// TIA Portal project "MPS1.1" (V16)

(* hardware
DEVICE "S7-1200 station_1"  S7-1200 Station
   slot 0: "Rack_0"  S7-1200 Rack  Rack  V1.0
   slot 1: "PLC_1"  CPU 1214C DC/DC/DC  6ES7 214-1AG40-0XB0  V4.4
   slot 2: "DI 8/DQ 8x24VDC_1"  6ES7 223-1BH32-0XB0  V2.0
*)

// ===== PLC "PLC_1"  CPU 1214C DC/DC/DC =====

VAR_GLOBAL   // PLC tag table "Default tag table"
   "System_Byte" AT %MB1 : Byte;
   "FirstScan" AT %M1.0 : Bool;
   "DiagStatusUpdate" AT %M1.1 : Bool;
   "AlwaysTRUE" AT %M1.2 : Bool;
   "AlwaysFALSE" AT %M1.3 : Bool;
   "Start NO" AT %I0.0 : Bool;
   "Stop NC" AT %I0.1 : Bool;
   "Reset NO" AT %I0.2 : Bool;
   "M/A Seletor" AT %I0.3 : Bool;
   "C2BG1" AT %I0.5 : Bool;
   "C2BG2" AT %I0.6 : Bool;
   "PART-AV1" AT %I0.7 : Bool;
   "C2BG3 NC" AT %I1.0 : Bool;
   "G1BG1 NO" AT %I1.1 : Bool;
   "G1BG2 NO" AT %I1.2 : Bool;
   "G1BG3 NC" AT %I1.3 : Bool;
   "Emergência NC" AT %I1.4 : Bool;
   "Pressostato NC" AT %I1.5 : Bool;
   "LED Start" AT %Q0.0 : Bool;
   "LED Reset" AT %Q0.1 : Bool;
   "Luz Q1" AT %Q0.2 : Bool;
   "Luz Q2" AT %Q0.3 : Bool;
   "Conv. anda p/ dir." AT %Q0.4 : Bool;
   "Conv. anda p/ esq." AT %Q0.5 : Bool;
   "Av. Cil. Alim." AT %Q0.6 : Bool;
   "Seletor Conv." AT %Q0.7 : Bool;
   "Válvula NC" AT %Q1.0 : Bool;
   "T1_STATUS" AT %M0.0 : Bool;
   "T2_STATUS" AT %M0.1 : Bool;
   "T3_STATUS" AT %M0.2 : Bool;
   "E1" AT %M0.3 : Bool;
   "E2" AT %M0.4 : Bool;
   "E3" AT %M0.5 : Bool;
   "E4" AT %M0.6 : Bool;
   "E5" AT %M0.7 : Bool;
   "E6" AT %M1.4 : Bool;
   "E7" AT %M1.5 : Bool;
   "E8" AT %M1.6 : Bool;
   "E9" AT %M1.7 : Bool;
   "E10" AT %M2.0 : Bool;
   "E11" AT %M2.1 : Bool;
   "E12" AT %M2.2 : Bool;
   "E13" AT %M2.3 : Bool;
   "E14" AT %M2.4 : Bool;
   "E15" AT %M2.5 : Bool;
   "E16" AT %M2.6 : Bool;
   "E17" AT %M2.7 : Bool;
   "E18" AT %M3.0 : Bool;
   "BIT.STOP" AT %M3.1 : Bool;
   "T4_STATUS" AT %M3.2 : Bool;
   "STATUS_E1" AT %M3.3 : Bool;
   "STATUS_E2" AT %M3.4 : Bool;
   "STATUS_E3" AT %M3.5 : Bool;
   "STATUS_E4" AT %M3.6 : Bool;
   "STATUS_E5" AT %M3.7 : Bool;
   "STATUS_E6" AT %M4.0 : Bool;
   "STATUS_E7" AT %M4.1 : Bool;
   "STATUS_E8" AT %M4.2 : Bool;
   "STATUS_E9" AT %M4.3 : Bool;
   "STATUS_E10" AT %M4.4 : Bool;
   "STATUS_E11" AT %M4.5 : Bool;
   "STATUS_E12" AT %M4.6 : Bool;
   "STATUS_E13" AT %M4.7 : Bool;
   "STATUS_E14" AT %M5.0 : Bool;
   "STATUS_E15" AT %M5.1 : Bool;
   "STATUS_E16" AT %M5.2 : Bool;
   "STATUS_E17" AT %M5.3 : Bool;
   "STATUS_E18" AT %M5.4 : Bool;
   "STATUS_E19" AT %M5.5 : Bool;
   "T5_STATUS" AT %M5.6 : Bool;
   "EStart_luzes" AT %M5.7 : Bool;
   "STATUS_ESTART" AT %M6.0 : Bool;
   "part-av1_status" AT %M6.1 : Bool;
END_VAR

// folder: System blocks/Program resources

DATA_BLOCK "T1"   // DB1
{ S7_Optimized_Access := 'TRUE' }
AUTHOR : Simatic
FAMILY : IEC
NAME : IEC_TMR
VERSION : 1.0
// stored: InstanceOfName IEC_TIMER
"IEC_TIMER"
BEGIN
END_DATA_BLOCK

DATA_BLOCK "T2"   // DB2
{ S7_Optimized_Access := 'TRUE' }
AUTHOR : Simatic
FAMILY : IEC
NAME : IEC_TMR
VERSION : 1.0
// stored: InstanceOfName IEC_TIMER
"IEC_TIMER"
BEGIN
END_DATA_BLOCK

DATA_BLOCK "T6"   // DB3
{ S7_Optimized_Access := 'TRUE' }
AUTHOR : Simatic
FAMILY : IEC
NAME : IEC_TMR
VERSION : 1.0
// stored: InstanceOfName IEC_TIMER
"IEC_TIMER"
BEGIN
END_DATA_BLOCK

DATA_BLOCK "T4"   // DB4
{ S7_Optimized_Access := 'TRUE' }
AUTHOR : Simatic
FAMILY : IEC
NAME : IEC_TMR
VERSION : 1.0
// stored: InstanceOfName IEC_TIMER
"IEC_TIMER"
BEGIN
END_DATA_BLOCK

DATA_BLOCK "T5"   // DB5
{ S7_Optimized_Access := 'TRUE' }
AUTHOR : Simatic
FAMILY : IEC
NAME : IEC_TMR
VERSION : 1.0
// stored: InstanceOfName IEC_TIMER
"IEC_TIMER"
BEGIN
END_DATA_BLOCK

DATA_BLOCK "Temporizador"   // DB7
{ S7_Optimized_Access := 'TRUE' }
AUTHOR : Simatic
FAMILY : IEC
NAME : IEC_TMR
VERSION : 1.0
// stored: InstanceOfName IEC_TIMER
"IEC_TIMER"
BEGIN
END_DATA_BLOCK

// folder: (top level)

FUNCTION "Main2" : Void   // FC1, LAD
{ S7_Optimized_Access := 'TRUE' }
VERSION : 0.1
BEGIN

REGION Network 1
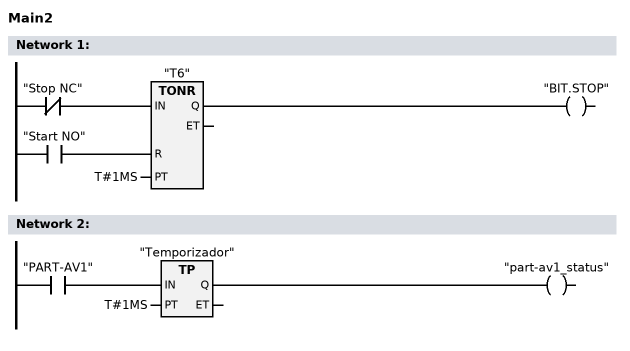
   "T6".TONR(IN := NOT "Stop NC", R := "Start NO", PT := T#1MS);
   "BIT.STOP" := "T6".Q;
END_REGION

REGION Network 2
   "Temporizador".TP(IN := "PART-AV1", PT := T#1MS);
   "part-av1_status" := "Temporizador".Q;
END_REGION
END_FUNCTION

ORGANIZATION_BLOCK "Main"   // OB1, LAD, ProgramCycle
TITLE = "Main Program Sweep (Cycle)"
{ S7_Optimized_Access := 'TRUE' }
VERSION : 0.1
   VAR_INPUT
      Initial_Call : Bool;   // Initial call of this OB
      Remanence : Bool;   // =True, if remanent data are available
   END_VAR
BEGIN

REGION Network 1
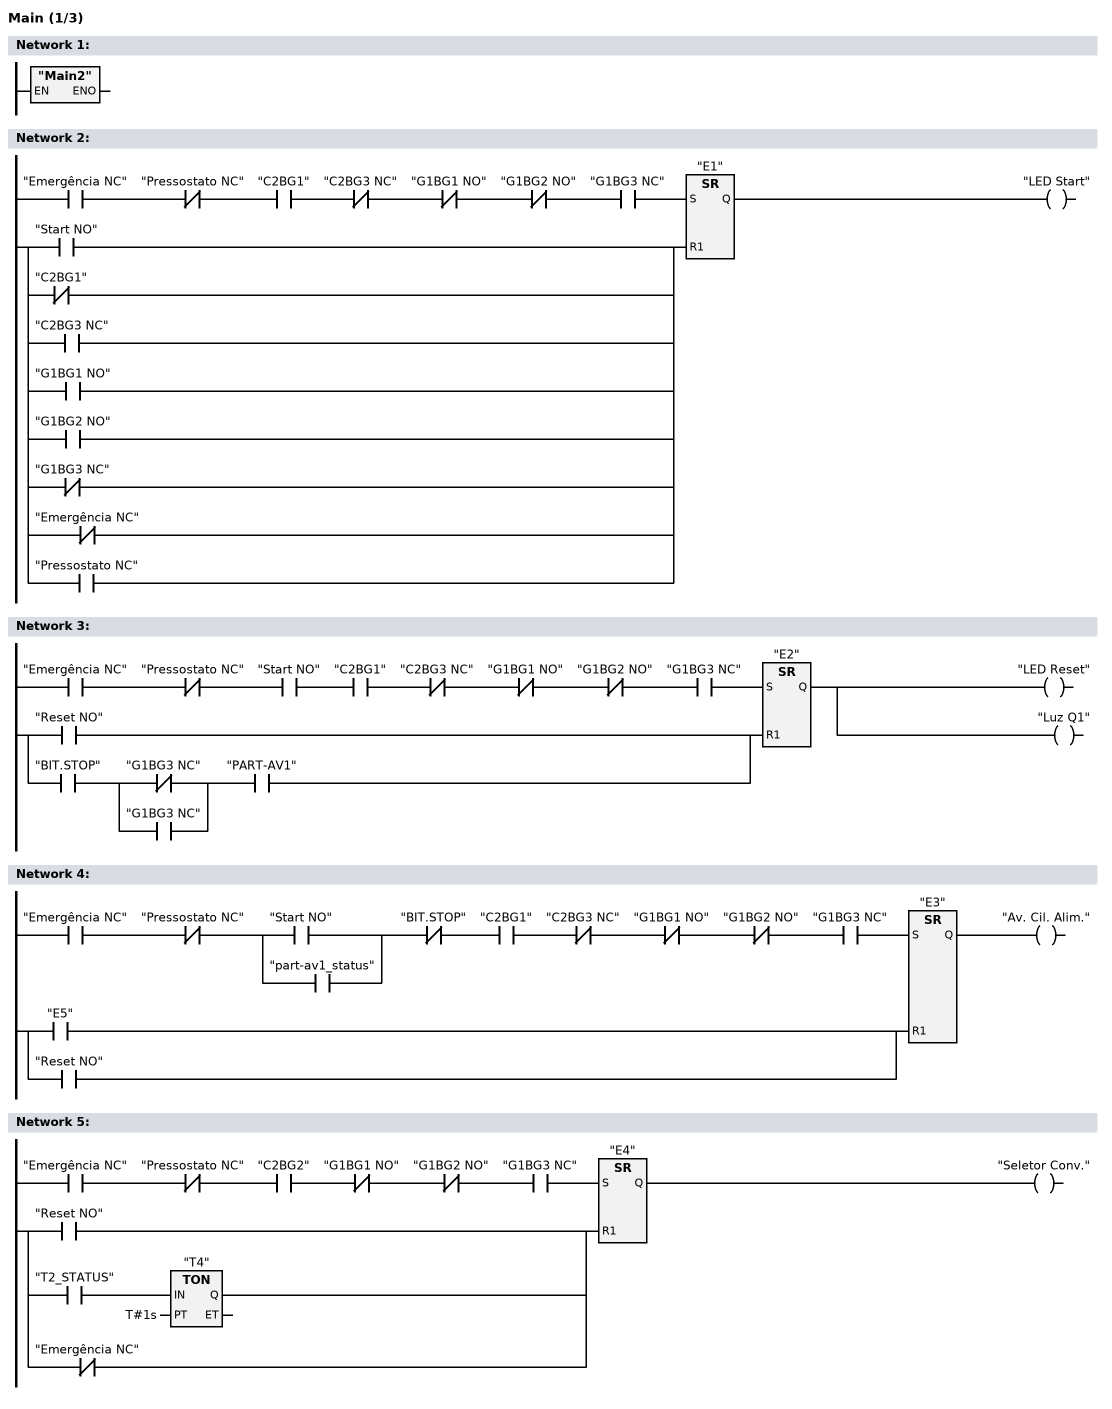
   RUNG wire#powerrail
      "Main2"()
   END_RUNG
   // the same network as SCL:
   "Main2"();
END_REGION

REGION Network 2
   RUNG wire#powerrail
      Contact( "Emergência NC" )
      I_Contact( "Pressostato NC" )
      Contact( "C2BG1" )
      I_Contact( "C2BG3 NC" )
      I_Contact( "G1BG1 NO" )
      I_Contact( "G1BG2 NO" )
      Contact( "G1BG3 NC" )
      S_SR(operand := "E1", r1 := wire#w1)
      Coil( "LED Start" )
   END_RUNG
   RUNG wire#powerrail
      Contact( "Start NO" )
   END_RUNG wire#w1
   RUNG wire#powerrail
      I_Contact( "C2BG1" )
   END_RUNG wire#w1
   RUNG wire#powerrail
      Contact( "C2BG3 NC" )
   END_RUNG wire#w1
   RUNG wire#powerrail
      Contact( "G1BG1 NO" )
   END_RUNG wire#w1
   RUNG wire#powerrail
      Contact( "G1BG2 NO" )
   END_RUNG wire#w1
   RUNG wire#powerrail
      I_Contact( "G1BG3 NC" )
   END_RUNG wire#w1
   RUNG wire#powerrail
      I_Contact( "Emergência NC" )
   END_RUNG wire#w1
   RUNG wire#powerrail
      Contact( "Pressostato NC" )
   END_RUNG wire#w1
   // the same network as SCL:
   IF "Emergência NC" AND NOT "Pressostato NC" AND "C2BG1" AND NOT "C2BG3 NC" AND NOT "G1BG1 NO" AND NOT "G1BG2 NO" AND "G1BG3 NC" THEN
       "E1" := TRUE;   // SR flip-flop
   END_IF;
   IF "Start NO" OR NOT "C2BG1" OR "C2BG3 NC" OR "G1BG1 NO" OR "G1BG2 NO" OR NOT "G1BG3 NC" OR NOT "Emergência NC" OR "Pressostato NC" THEN
       "E1" := FALSE;
   END_IF;
   "LED Start" := "E1";
END_REGION

REGION Network 3
   RUNG wire#powerrail
      Contact( "Emergência NC" )
      I_Contact( "Pressostato NC" )
      Contact( "Start NO" )
      Contact( "C2BG1" )
      I_Contact( "C2BG3 NC" )
      I_Contact( "G1BG1 NO" )
      I_Contact( "G1BG2 NO" )
      Contact( "G1BG3 NC" )
      S_SR(operand := "E2", r1 := wire#w3)
      wire#w4
      Coil( "LED Reset" )
   END_RUNG
   RUNG wire#powerrail
      Contact( "Reset NO" )
   END_RUNG wire#w3
   RUNG wire#powerrail
      Contact( "BIT.STOP" )
      wire#w1
      I_Contact( "G1BG3 NC" )
      wire#w2
      Contact( "PART-AV1" )
   END_RUNG wire#w3
   RUNG wire#w1
      Contact( "G1BG3 NC" )
   END_RUNG wire#w2
   RUNG wire#w4
      Coil( "Luz Q1" )
   END_RUNG
   // the same network as SCL:
   IF "Emergência NC" AND NOT "Pressostato NC" AND "Start NO" AND "C2BG1" AND NOT "C2BG3 NC" AND NOT "G1BG1 NO" AND NOT "G1BG2 NO" AND "G1BG3 NC" THEN
       "E2" := TRUE;   // SR flip-flop
   END_IF;
   IF "Reset NO" OR ("BIT.STOP" AND (NOT "G1BG3 NC" OR "G1BG3 NC") AND "PART-AV1") THEN
       "E2" := FALSE;
   END_IF;
   "LED Reset" := "E2";
   "Luz Q1" := "E2";
END_REGION

REGION Network 4
   RUNG wire#powerrail
      Contact( "Emergência NC" )
      I_Contact( "Pressostato NC" )
      wire#w1
      Contact( "Start NO" )
      wire#w2
      I_Contact( "BIT.STOP" )
      Contact( "C2BG1" )
      I_Contact( "C2BG3 NC" )
      I_Contact( "G1BG1 NO" )
      I_Contact( "G1BG2 NO" )
      Contact( "G1BG3 NC" )
      S_SR(operand := "E3", r1 := wire#w3)
      Coil( "Av. Cil. Alim." )
   END_RUNG
   RUNG wire#w1
      Contact( "part-av1_status" )
   END_RUNG wire#w2
   RUNG wire#powerrail
      Contact( "E5" )
   END_RUNG wire#w3
   RUNG wire#powerrail
      Contact( "Reset NO" )
   END_RUNG wire#w3
   // the same network as SCL:
   IF "Emergência NC" AND NOT "Pressostato NC" AND ("Start NO" OR "part-av1_status") AND NOT "BIT.STOP" AND "C2BG1" AND NOT "C2BG3 NC" AND NOT "G1BG1 NO" AND NOT "G1BG2 NO" AND "G1BG3 NC" THEN
       "E3" := TRUE;   // SR flip-flop
   END_IF;
   IF "E5" OR "Reset NO" THEN "E3" := FALSE; END_IF;
   "Av. Cil. Alim." := "E3";
END_REGION

REGION Network 5
   "T4".TON(IN := "T2_STATUS", PT := T#1s);
   IF "Emergência NC" AND NOT "Pressostato NC" AND "C2BG2" AND NOT "G1BG1 NO" AND NOT "G1BG2 NO" AND "G1BG3 NC" THEN
       "E4" := TRUE;   // SR flip-flop
   END_IF;
   IF "Reset NO" OR "T4".Q OR NOT "Emergência NC" THEN "E4" := FALSE; END_IF;
   "Seletor Conv." := "E4";
END_REGION

REGION Network 6
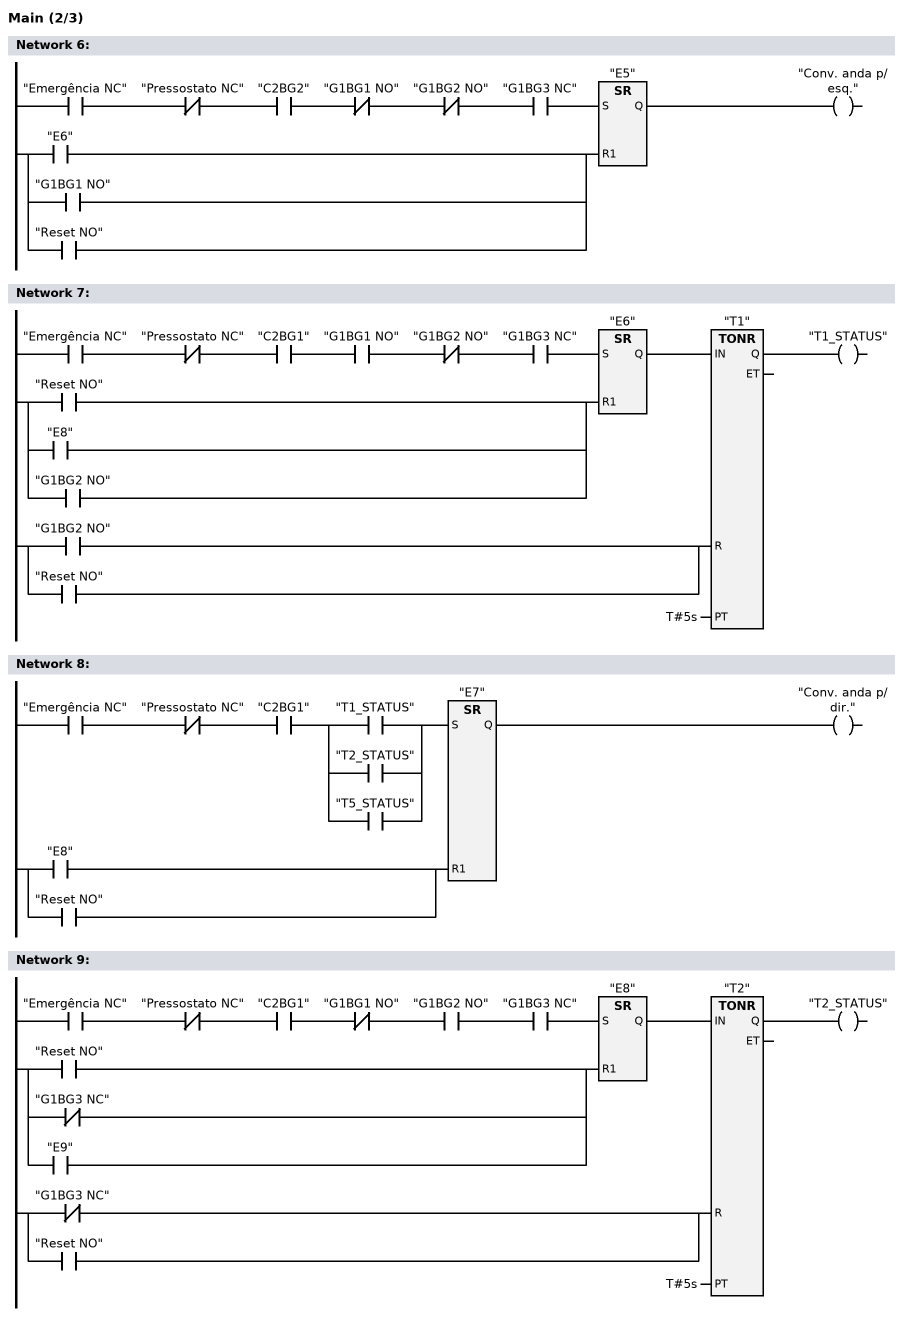
   RUNG wire#powerrail
      Contact( "Emergência NC" )
      I_Contact( "Pressostato NC" )
      Contact( "C2BG2" )
      I_Contact( "G1BG1 NO" )
      I_Contact( "G1BG2 NO" )
      Contact( "G1BG3 NC" )
      S_SR(operand := "E5", r1 := wire#w1)
      Coil( "Conv. anda p/ esq." )
   END_RUNG
   RUNG wire#powerrail
      Contact( "E6" )
   END_RUNG wire#w1
   RUNG wire#powerrail
      Contact( "G1BG1 NO" )
   END_RUNG wire#w1
   RUNG wire#powerrail
      Contact( "Reset NO" )
   END_RUNG wire#w1
   // the same network as SCL:
   IF "Emergência NC" AND NOT "Pressostato NC" AND "C2BG2" AND NOT "G1BG1 NO" AND NOT "G1BG2 NO" AND "G1BG3 NC" THEN
       "E5" := TRUE;   // SR flip-flop
   END_IF;
   IF "E6" OR "G1BG1 NO" OR "Reset NO" THEN "E5" := FALSE; END_IF;
   "Conv. anda p/ esq." := "E5";
END_REGION

REGION Network 7
   IF "Emergência NC" AND NOT "Pressostato NC" AND "C2BG1" AND "G1BG1 NO" AND NOT "G1BG2 NO" AND "G1BG3 NC" THEN
       "E6" := TRUE;   // SR flip-flop
   END_IF;
   IF "Reset NO" OR "E8" OR "G1BG2 NO" THEN "E6" := FALSE; END_IF;
   "T1".TONR(IN := "E6", R := "G1BG2 NO" OR "Reset NO", PT := T#5s);
   "T1_STATUS" := "T1".Q;
END_REGION

REGION Network 8
   RUNG wire#powerrail
      Contact( "Emergência NC" )
      I_Contact( "Pressostato NC" )
      Contact( "C2BG1" )
      wire#w1
      Contact( "T1_STATUS" )
      wire#w2
      S_SR(operand := "E7", r1 := wire#w3)
      Coil( "Conv. anda p/ dir." )
   END_RUNG
   RUNG wire#w1
      Contact( "T2_STATUS" )
   END_RUNG wire#w2
   RUNG wire#w1
      Contact( "T5_STATUS" )
   END_RUNG wire#w2
   RUNG wire#powerrail
      Contact( "E8" )
   END_RUNG wire#w3
   RUNG wire#powerrail
      Contact( "Reset NO" )
   END_RUNG wire#w3
   // the same network as SCL:
   IF "Emergência NC" AND NOT "Pressostato NC" AND "C2BG1" AND ("T1_STATUS" OR "T2_STATUS" OR "T5_STATUS") THEN
       "E7" := TRUE;   // SR flip-flop
   END_IF;
   IF "E8" OR "Reset NO" THEN "E7" := FALSE; END_IF;
   "Conv. anda p/ dir." := "E7";
END_REGION

REGION Network 9
   IF "Emergência NC" AND NOT "Pressostato NC" AND "C2BG1" AND NOT "G1BG1 NO" AND "G1BG2 NO" AND "G1BG3 NC" THEN
       "E8" := TRUE;   // SR flip-flop
   END_IF;
   IF "Reset NO" OR NOT "G1BG3 NC" OR "E9" THEN "E8" := FALSE; END_IF;
   "T2".TONR(IN := "E8", R := NOT "G1BG3 NC" OR "Reset NO", PT := T#5s);
   "T2_STATUS" := "T2".Q;
END_REGION

REGION Network 10
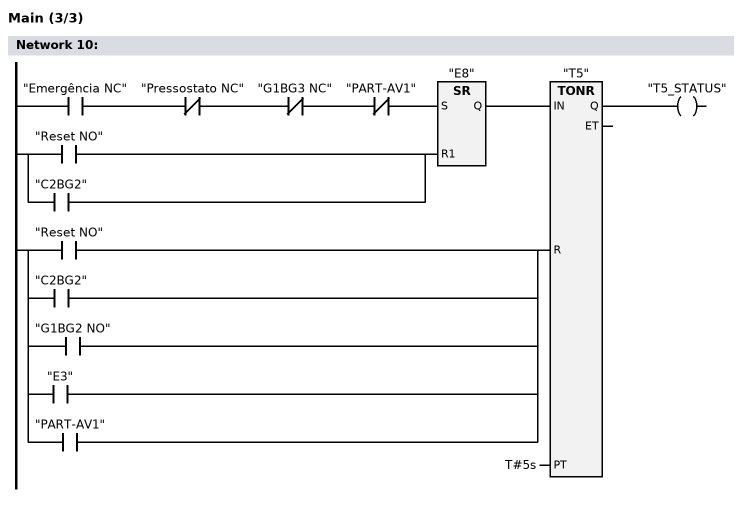
   IF "Emergência NC" AND NOT "Pressostato NC" AND NOT "G1BG3 NC" AND NOT "PART-AV1" THEN
       "E8" := TRUE;   // SR flip-flop
   END_IF;
   IF "Reset NO" OR "C2BG2" THEN "E8" := FALSE; END_IF;
   "T5".TONR(IN := "E8", R := "Reset NO" OR "C2BG2" OR "G1BG2 NO" OR "E3" OR "PART-AV1", PT := T#5s);
   "T5_STATUS" := "T5".Q;
END_REGION
END_ORGANIZATION_BLOCK